(* IEC 61131-3 sources: AutomationStudio/DystrybucjaWodySekwencer, 3 files *)

(* ---- Types.typ ---- *)
TYPE
	SterowanieTyp :
		(
		AWARIA := 5, (*oBSLUGA AWARII -> gorące styki stycznika pompy, suchobieg - przepływ poniżej minimum*)
		WYBIEG := 4, (*Procedura zatrzymywania -> spdek ciśnienia poniżej minimum i przepływu poniżej min*)
		POMPOWANIE := 3, (*Normalnia praca, utrzymywanie ciśnienia powyżej wiekszgo niż min i przepływu wiekszego niż min*)
		INITIAL := 1, (*Czekanie na rozruch*)
		ROZRUCH := 2 (*Porcedura rozruchowa *)
	);

	PumpTyp : STRUCT
		doPompa : BOOL; (*Wysterowanie stycznika pompy*)
		diTermik : BOOL := TRUE; (*TERMOSTAT wykrywający gorące styki stycznika*)
		diCisnienieMin : BOOL; (*presostat wykrywający ciśnienie minimalne*)
		diCisnienieMax : BOOL :=TRUE;
		diPrzeplywMin : BOOL; (*Czujnik wykrywajacy przeplyw minimalny*)
		diPrzeplywMax : BOOL :=TRUE; (*Czujnik wykrywajacy przeplyw maksymalny*)
	END_STRUCT;

	OperatorTyp : STRUCT
		diStart : BOOL; (*Przycisk start NO*)
		diStop : BOOL := TRUE; (*Przycisk STOP NC*)
		diEStop : BOOL := TRUE; (*Wyłącznik bezpieczenstaw nc*)
		doSystemAktywny : BOOL; (*Lampka system aktywny*)
		doAwaria : BOOL; (*Lampka awaria*)
		diKasujAwaria : BOOL; (*Przycisk kasowania awarii*)
	END_STRUCT;

	DystrybucjaCieczyTyp : STRUCT
		Pompa : PumpTyp;
		Operator : OperatorTyp;
	END_STRUCT;

	SystemParTyp : STRUCT
		uiCzasSensor : ARRAY[0..9] OF REAL;(*Czas aktywności sensora wykrywającego usterkę np. termik [sekundy]*)
		uiCzasWybieg : ARRAY[0..9] OF REAL;(*Czas aktywności sensora wykrywającego usterkę np. termik [sekundy]*)
		uiCzasRozruch : ARRAY[0..9] OF REAL;
	END_STRUCT;

END_TYPE

(* ---- Main.st ---- *)
PROGRAM _INIT
	(* Insert code here *)
	 Sterowanie:= INITIAL;
END_PROGRAM

PROGRAM _CYCLIC
	(* Maszyna stanu do systemu dystrybucji wody *)

	CASE Sterowanie OF
		INITIAL:
			FOR i:=0 TO 9 DO
				ZegarTON[i].IN:=FALSE; (*KAsowanie stanmów zegara*)
				ZegarTON[i]();
			END_FOR;

			DystrybucjaCieczy.Operator.doSystemAktywny:=(DystrybucjaCieczy.Operator.diStart OR
			DystrybucjaCieczy.Operator.doSystemAktywny) AND DystrybucjaCieczy.Operator.diEStop
			AND DystrybucjaCieczy.Operator.diStop;

			IF (DystrybucjaCieczy.Operator.doSystemAktywny AND DystrybucjaCieczy.Pompa.diTermik) THEN
				Sterowanie:=ROZRUCH;
			END_IF;

			IF (DystrybucjaCieczy.Operator.doSystemAktywny AND NOT(DystrybucjaCieczy.Pompa.diTermik)) THEN
				(*Wpisujemy indeks do tablicy alarmow i przekazujemy do bazy danych*)
				Sterowanie:=AWARIA;
			END_IF;

		ROZRUCH:
			ZegarTON[1].IN:=NOT(DystrybucjaCieczy.Pompa.diTermik);
			ZegarTON[1].PT:=REAL_TO_TIME(DystrybucjaCieczyPar.uiCzasSensor[0]*1000);
			ZegarTON[1]();

			ZegarTON[2].IN:=TRUE;
			ZegarTON[2].PT:=REAL_TO_TIME(DystrybucjaCieczyPar.uiCzasSensor[0]*1000);
			ZegarTON[2]();

			DystrybucjaCieczy.Pompa.doPompa:=TRUE; //akcja

			IF (DystrybucjaCieczy.Pompa.diCisnienieMin AND DystrybucjaCieczy.Pompa.diPrzeplywMin) THEN
				Sterowanie:=POMPOWANIE;
			END_IF;
			IF NOT(DystrybucjaCieczy.Operator.diStop) THEN
				Sterowanie:= WYBIEG;
			END_IF;
			IF NOT(DystrybucjaCieczy.Operator.diStop) THEN
				Sterowanie:=AWARIA;
			END_IF;
			IF ZegarTON[1].Q THEN
				(*Wprowadz indeks DO tablicy alarmów*)
				Sterowanie:=AWARIA;
			END_IF;
			IF ZegarTON[2].Q THEN
				(*Wprowadz indeks do tablicy alarmów*)
				Sterowanie:=AWARIA;
			END_IF;

		POMPOWANIE:
			ZegarTON[1].IN:=NOT(DystrybucjaCieczy.Pompa.diTermik);
			ZegarTON[1].PT:=REAL_TO_TIME(DystrybucjaCieczyPar.uiCzasSensor[1]*1000);
			ZegarTON[1]();

			ZegarTON[3].IN:=NOT(DystrybucjaCieczy.Pompa.diCisnienieMin);
			ZegarTON[3].PT:=REAL_TO_TIME(DystrybucjaCieczyPar.uiCzasSensor[3]*1000);
			ZegarTON[3]();

			ZegarTON[4].IN:=NOT(DystrybucjaCieczy.Pompa.diPrzeplywMin);
			ZegarTON[4].PT:=REAL_TO_TIME(DystrybucjaCieczyPar.uiCzasSensor[4]*1000);
			ZegarTON[4]();

			IF NOT(DystrybucjaCieczy.Operator.diStop) THEN
				Sterowanie:=WYBIEG;
			END_IF;
			IF NOT(DystrybucjaCieczy.Operator.diStop) THEN
				Sterowanie:=AWARIA;
			END_IF;
			IF ZegarTON[1].Q THEN
				(*Wprowadz indeks DO tablicy alarmów*)
				Sterowanie:=AWARIA;
			END_IF;
			IF ZegarTON[3].Q THEN
				(*Wprowadz indeks DO tablicy alarmów*)
				Sterowanie:=AWARIA;
			END_IF;
			IF ZegarTON[4].Q THEN
				(*Wprowadz indeks DO tablicy alarmów*)
				Sterowanie:=AWARIA;
			END_IF;
		WYBIEG:
			DystrybucjaCieczy.Pompa.doPompa:=FALSE;

			ZegarTON[1].IN:=NOT(DystrybucjaCieczy.Pompa.diTermik);
			ZegarTON[1].PT:=REAL_TO_TIME(DystrybucjaCieczyPar.uiCzasSensor[0]*1000);
			ZegarTON[1]();

			IF (NOT(DystrybucjaCieczy.Pompa.diCisnienieMin) AND NOT(DystrybucjaCieczy.Pompa.diPrzeplywMin)) THEN
				DystrybucjaCieczy.Operator.doSystemAktywny:=FALSE;
				Sterowanie:=INITIAL;
			END_IF;
			IF NOT(DystrybucjaCieczy.Operator.diStop) THEN
				(*Wprowadz indeks DO tablicy alarmów*)
				Sterowanie:=AWARIA;
			END_IF;
			IF ZegarTON[1].Q THEN
				(*Wprowadz indeks DO tablicy alarmów*)
				Sterowanie:=AWARIA;
			END_IF;

		AWARIA:
			DystrybucjaCieczy.Operator.doSystemAktywny:=FALSE;
			DystrybucjaCieczy.Pompa.doPompa:=FALSE;
			ZegarTON[0].IN:=NOT(ZegarTON[0].Q);
			ZegarTON[0].PT:=T#300ms;
			ZegarTON[0]();
			DystrybucjaCieczy.Operator.doAwaria:=DystrybucjaCieczy.Operator.doAwaria XOR ZegarTON[0].Q;
			IF (DystrybucjaCieczy.Operator.diKasujAwaria AND DystrybucjaCieczy.Pompa.diTermik AND DystrybucjaCieczy.Operator.diStop) THEN
				DystrybucjaCieczy.Operator.doAwaria:=FALSE;
				(*Potwierdzamy alarm i przekazujemy do bazy danych*)
				Sterowanie:=INITIAL;
			END_IF

	END_CASE;

END_PROGRAM

PROGRAM _EXIT
	(* Insert code here *)

END_PROGRAM

(* ---- Variables.var ---- *)
VAR
	i : INT;
	Sterowanie : SterowanieTyp;
	DystrybucjaCieczy : DystrybucjaCieczyTyp;
	ZegarTON : ARRAY[0..10] OF TON;
END_VAR
VAR RETAIN
	DystrybucjaCieczyPar : SystemParTyp; (*Parametry podtrzymywane w pamięci flash lub bateryjnie*)
END_VAR
